{region '#Template'}
	{attribute 'Category' := 'General'}
	{attribute 'Version' := '0.0.2.0'}
	{attribute 'Tags' := 'Trade, Plant, General'}
	{attribute 'Description' := 'Aufruf der Anlagen des Gewerks Allgemein	// Calling the plants of the trade general'}
{endregion}
FUNCTION_BLOCK FB_BA_General EXTENDS FB_BA_View
VAR_INPUT
	fTWth			: REAL;	//	Weather temperature
END_VAR
VAR_INPUT CONSTANT
	// [Sample] "Implementieren lokaler(!) Informationen und Funktionen"
	// Mit "lokal" ist gemeint dass es in einem Projekt mit mehreren SPS'en eine "Master-SPS" gibt, die Informationen (Sollwerte und Zustände) bereitstellt.
	// Betreiber greifen an dieser zentralen Stelle auf Informationen zu, welche dann von der "Master-SPS" an die "Slave-SPS" verteilt werden.
	IFP					: FB_BA_IFP;											 
	EvtGroups			: FB_BA_EvtGroups;											 
	Settings			: FB_BA_Settings;
	Cabinet				: FB_BA_ControlCabinet;				 
	BuildingGlobal		: FB_BA_BuildingGlobal;

	WeatherStation		: FB_BA_RawSubscriber;
	stWeatherStation	: ST_BA_WeatherStation;	
END_VAR

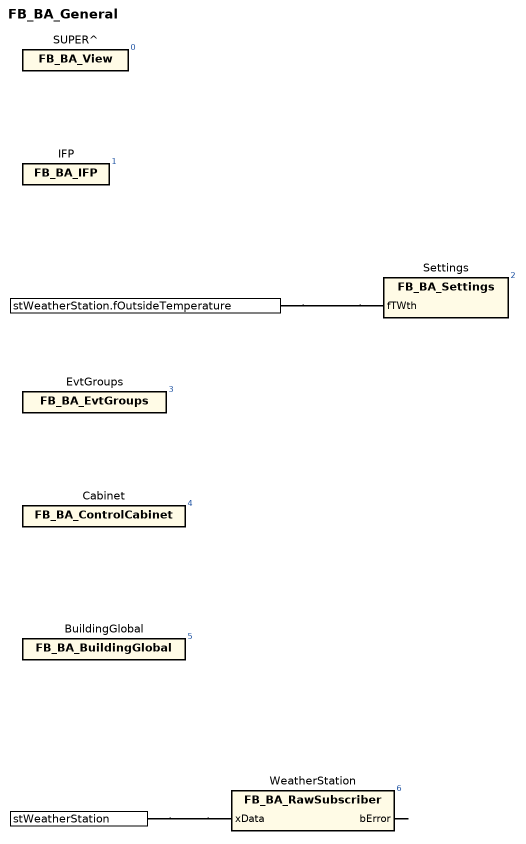
SUPER^(); // FB_BA_View
IFP(); // FB_BA_IFP
Settings(fTWth := stWeatherStation.fOutsideTemperature); // FB_BA_Settings
EvtGroups(); // FB_BA_EvtGroups
Cabinet(); // FB_BA_ControlCabinet
BuildingGlobal(); // FB_BA_BuildingGlobal
WeatherStation(xData := stWeatherStation); // FB_BA_RawSubscriber

METHOD FB_init : BOOL
VAR_INPUT
	bInitRetains : BOOL; // if TRUE, the retain variables are initialized (warm start / cold start)
	bInCopyCode : BOOL;  // if TRUE, the instance afterwards gets moved into the copy code (online change)
END_VAR
IFP.iParent						:= THIS^;	
IFP.sObjectName					:= TextPlants.Information_focal_point_sObjectname;
IFP.sDescription				:= TextPlants.Information_focal_point_sDescription;
IFP.eDPADMode					:= E_BA_DPADMode.eInclude;		

EvtGroups.iParent				:= THIS^;	
EvtGroups.sObjectName			:= TextPlants.EventGroups_sObjectName;
EvtGroups.sDescription			:= TextPlants.EventGroups_sDescription;
EvtGroups.eDPADMode				:= E_BA_DPADMode.eInclude;									

Settings.iParent				:= THIS^;										 
Settings.sObjectName			:= TextPlants.Settings_sObjectName;
Settings.sDescription			:= TextPlants.Settings_sDescription;
Settings.eDPADMode				:= E_BA_DPADMode.eInclude;

Cabinet.iParent					:= THIS^;	
Cabinet.sObjectName				:= TextPlants.Control_cabinet_sObjectName;
Cabinet.sDescription			:= TextPlants.Control_cabinet_sDescription;									 
Cabinet.eDPADMode				:= E_BA_DPADMode.eInclude;
				 
BuildingGlobal.iParent			:= THIS^;	
BuildingGlobal.sObjectName		:= TextPlants.Global_Building_Data_sObjectName;														 
BuildingGlobal.sDescription		:= TextPlants.Global_Building_Data_sDescription;														 
BuildingGlobal.eDPADMode		:= E_BA_DPADMode.eInclude;

WeatherStation.Subject			:= Site.WeatherStation_Subject;
WeatherStation.sTarget			:= Site.WeatherStation_NetId;
END_METHOD

END_FUNCTION_BLOCK

(* stored: Version 1.1.0.1, ProductVersion 3.1.4024.6
   POU FB_BA_General: Id {4f3eddb1-0308-4e4b-a4e2-7cdc9ca29c8b}, SpecialFunc None
   Method FB_init: Id {63ef2833-b0ed-49d1-b83a-d3b3ee61d402} *)
